{attribute 'GeneratedUsingTerminal: EK1100-0000-0018'}
{attribute addProperty BoxType "EK1100-0000-0018"}
{attribute addProperty Id "Term_330_EK1122Term_330_EK1122_0EDE60FE40Term_335_EL2008EL2008_E2806B9511Term_336_EL2008EL2008_E2806B9511"}
{attribute addProperty CRC "3952060993"}
{attribute addProperty Size "62"}
{attribute addProperty Name "Term 307 (EK1100)"}
TYPE Term_307_EK1100_EB8FAA41 EXTENDS EK1100_1FC0878B :
STRUCT
	{attribute addProperty Name "Term 330 (EK1122)"}
	{attribute addProperty PreviousPort "Term 307 (EK1100) : B"}
	{attribute addProperty SyncUnit "default"}
	Term_330_EK1122 : Term_330_EK1122_0EDE60FE;
	{attribute addProperty Name "Term 335 (EL2008)"}
	{attribute addProperty PreviousPort "Term 330 (EK1122) : C"}
	{attribute addProperty SyncUnit "default"}
	Term_335_EL2008 : EL2008_E2806B95;
	{attribute addProperty Name "Term 336 (EL2008)"}
	{attribute addProperty PreviousPort "Term 335 (EL2008) : B"}
	{attribute addProperty SyncUnit "default"}
	Term_336_EL2008 : EL2008_E2806B95;
END_STRUCT
END_TYPE

(* stored: Version 1.2.0.0, ProductVersion 3.1.4024.11
   DUT Term_307_EK1100_EB8FAA41: Id {d46fe168-1655-49f7-99c4-c77d69bb177b} *)
